FUNCTION_BLOCK TEST_MODEL
  {SET_ATTRIBUTE(OpcUa, SERVICE)}
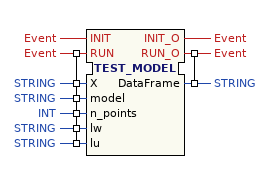
  EVENT_INPUT
    INIT;
    RUN WITH X, model, n_points, lw, lu; {SET_ATTRIBUTE(OpcUa, Method)}
  END_EVENT
  EVENT_OUTPUT
    INIT_O;
    RUN_O WITH DataFrame;
  END_EVENT
  VAR_INPUT
    X : STRING; {SET_ATTRIBUTE(OpcUa, Variable.RUN)}
    model : STRING; {SET_ATTRIBUTE(OpcUa, Variable.RUN)}
    n_points : INT; {SET_ATTRIBUTE(OpcUa, Variable.RUN)}
    lw : STRING; {SET_ATTRIBUTE(OpcUa, Variable.RUN)}
    lu : STRING; {SET_ATTRIBUTE(OpcUa, Variable.RUN)}
  END_VAR
  VAR_OUTPUT
    DataFrame : STRING; {SET_ATTRIBUTE(OpcUa, Variable.RUN)}
  END_VAR
END_FUNCTION_BLOCK
